(* IEC 61131-3 sources: repolevel_ST_code_completion/extract_code/轴控/FB105_轴控制集/FC11_设备状态, 3 files *)

(* ---- A03_气缸状态.st ---- *)
IF DI_取料上下气缸原点 AND DI_入料纠偏气缸原点 AND DI_翻板气缸原点 AND DI_左A包底气缸原点 AND DI_右B包底气缸原点 AND
	DI_上包底气缸原点 AND DI_出料推盒气缸原点 AND DI_包盒口升降气缸原点 AND DI_包盒口下压气缸原点 AND DI_推底板气缸原点 AND
	 DI_翻底板气缸原点 AND DI_模组吸底板气缸原点 THEN
	 b所有气缸原位OK:=TRUE;
	 ELSE
	 b所有气缸原位OK:=FALSE;
END_IF

IF NOT DO_取料气缸 AND NOT DO_纠偏气缸 AND NOT DO_挡料定位气缸 AND NOT DO_翻板气缸 AND NOT DO_侧压紧气缸 AND NOT DO_左A包底气缸 AND
	NOT DO_右B包底气缸 AND NOT DO_上包底气缸 AND NOT DO_下包底气缸 AND NOT DO_出料推盒气缸 AND NOT DO_包盒口升降气缸 AND
	NOT DO_包盒口下压气缸 AND NOT DO_翻底板气缸 AND NOT DO_推底板气缸 AND NOT DO_模组吸底板气缸 AND NOT DO_包边纠偏上下气缸 AND
	NOT DO_包边纠偏左右气缸 AND NOT DO_包边压料气缸 AND NOT DO_折边上托气缸 AND NOT DO_包边铲边气缸 AND NOT DO_吸底板真空 AND
	NOT DO_取面板真空 AND NOT DO_A模吸底板真空 AND NOT DO_A模吸面板真空 AND NOT DO_B模吸底板真空 AND NOT DO_B模吸面板真空 THEN
	b所有气缸关闭OK:=TRUE;
	ELSE
	b所有气缸关闭OK:=FALSE;
END_IF

(* ---- A04_初始化.st ---- *)
TON0(IN:= HMI_b初始化, PT:= T#3S, Q=> , ET=> );
TON1(IN:= HMI_b初始化, PT:= T#2S, Q=> , ET=> );
R_TRIG0(CLK:= TON0.Q AND b所有伺服使能OK AND b所有伺服总线通讯OK AND NOT b设备报警 AND b非急停手动模式 AND NOT b设备初始化中, Q=> );
R_TRIG1(CLK:= TON1.Q AND b所有伺服使能OK AND b所有伺服总线通讯OK AND NOT b设备报警 AND b非急停手动模式 AND NOT b设备初始化中, Q=> );

IF R_TRIG1.Q THEN
	b轴控初始化:=TRUE;
END_IF
TON4(IN:= b轴控初始化, PT:= T#0.3S, Q=> , ET=> );
IF TON4.Q THEN
	b轴控初始化:=FALSE;
END_IF

IF NOT DI_急停按钮 THEN
	i初始化步:=0;
	b设备初始化中:=FALSE;
	b调模A轴回零触发:=FALSE;
	b调模B轴回零触发:=FALSE;
	b送面料轴回零触发:=FALSE;
	b取面料轴回零触发:=FALSE;
	b横移A轴回零触发:=FALSE;
	b升降A轴回零触发:=FALSE;
	b横移B轴回零触发:=FALSE;
	b升降B轴回零触发:=FALSE;
	b出盒轴回零触发:=FALSE;
	b铲灰板轴回零触发:=FALSE;
	b包面纸轴回零触发:=FALSE;
	b上包底轴回零触发:=FALSE;
	b折边轴回零触发:=FALSE;
END_IF

CASE i初始化步 OF
	0:
	IF R_TRIG0.Q THEN
		b设备初始化中:=TRUE;
		i初始化步:=1;
	END_IF

	1:
	IF b设备初始化中 THEN
		b自动运行:=FALSE; b自动互锁:=FALSE;
		TON2(IN:= TRUE, PT:= T#0.2S, Q=> , ET=> );
		IF TON2.Q THEN
			TON2(IN:= FALSE,  );
			i初始化步:=5;
		END_IF

	END_IF

	5:

	IF b设备初始化中 THEN
		DO_取料气缸:=FALSE; DO_纠偏气缸:=FALSE; DO_挡料定位气缸:=FALSE; DO_翻板气缸:=FALSE; DO_侧压紧气缸:=FALSE;
		DO_左A包底气缸:=FALSE; DO_右B包底气缸:=FALSE; DO_上包底气缸:=FALSE; DO_下包底气缸:=FALSE; DO_出料推盒气缸:=FALSE;
		DO_包盒口升降气缸:=FALSE; DO_包盒口下压气缸:=FALSE; DO_翻底板气缸:=FALSE; DO_推底板气缸:=FALSE; DO_模组吸底板气缸:=FALSE;
		DO_包边纠偏上下气缸:=FALSE; DO_包边纠偏左右气缸:=FALSE; DO_包边压料气缸:=FALSE; DO_折边上托气缸:=FALSE;
        DO_包边铲边气缸:=FALSE; DO_吸底板真空:=FALSE; DO_取面板真空:=FALSE; DO_A模吸底板真空:=FALSE; DO_A模吸面板真空:=FALSE;
		DO_B模吸底板真空:=FALSE; DO_B模吸面板真空:=FALSE; DO_真空泵:=FALSE; DO_出料皮带电机:=FALSE;
		IF b所有气缸原位OK AND b所有气缸关闭OK THEN
			i初始化步:=10;
		END_IF
	END_IF

	10:
	IF b设备初始化中 THEN
		b调模A轴回零触发:=TRUE;
		b调模B轴回零触发:=TRUE;
		b送面料轴回零触发:=TRUE;
		b取面料轴回零触发:=TRUE;
		b横移A轴回零触发:=TRUE;
		b升降A轴回零触发:=TRUE;
		b横移B轴回零触发:=TRUE;
		b升降B轴回零触发:=TRUE;
		b出盒轴回零触发:=TRUE;
		b铲灰板轴回零触发:=TRUE;
		b包面纸轴回零触发:=TRUE;
		b上包底轴回零触发:=TRUE;
		b折边轴回零触发:=TRUE;
		TON3(IN:= TRUE, PT:= T#0.2S, Q=> , ET=> );
		IF TON3.Q AND b所有伺服静止中 THEN
			b调模A轴回零触发:=FALSE;
		    b调模B轴回零触发:=FALSE;
		    b送面料轴回零触发:=FALSE;
		    b取面料轴回零触发:=FALSE;
		    b横移A轴回零触发:=FALSE;
		    b升降A轴回零触发:=FALSE;
		    b横移B轴回零触发:=FALSE;
		    b升降B轴回零触发:=FALSE;
		    b出盒轴回零触发:=FALSE;
		    b铲灰板轴回零触发:=FALSE;
		    b包面纸轴回零触发:=FALSE;
		    b上包底轴回零触发:=FALSE;
		    b折边轴回零触发:=FALSE;
			TON3(IN:= FALSE,  );
			i初始化步:=15;
		END_IF

	END_IF

	15:
	IF b设备初始化中 THEN
		b设备初始化中:=FALSE;
		i初始化步:=0;
	END_IF
END_CASE

(* ---- FB11_设备状态.st ---- *)
PROGRAM FC11_设备状态
VAR
	fb_bFristScan: TON;

	TON0: TON;
	TON1: TON;
	TON2: TON;
	TON3: TON;
	TON4: TON;

	i初始化步: INT;

	R_TRIG0: R_TRIG;
	R_TRIG1: R_TRIG;

END_VAR

(*IO功能启用*)
//NET_IO_Cmd(SysWarnID:= , bError=> , nErrorID=> );

(*子程序调用*)
A01_输入映射();

A02_输出映射();

A03_气缸状态();

A04_初始化();

(*开机初始化*)
fb_bFristScan(IN:= b常闭, PT:= T#1S, Q=> , ET=> );
IF TIME_TO_REAL(fb_bFristScan.ET)>500 AND TIME_TO_REAL(fb_bFristScan.ET)<600 THEN
	b开机初始化:=TRUE;
	ELSE
	b开机初始化:=FALSE;
END_IF

IF NOT b常通 THEN
	b开机第一次启动:=TRUE;
	ELSE
	b开机第一次启动:=FALSE;
END_IF
IF b开机第一次启动 OR b常通 THEN
	b常通:=TRUE;
	ELSE
	b常通:=FALSE;
END_IF
(*
IF EtherCAT_Master_Leadshine.xConfigFinished AND EtherCAT_Master_Leadshine.xDistributedClockInSync AND
   NOT EtherCAT_Master_Leadshine.xError AND NOT b常闭 THEN
	b开机初始化:=TRUE;
	ELSE
	b开机初始化:=FALSE;
END_IF
*)

(*状态判定*)
IF DI_急停按钮 AND NOT HMI_b手动模式0自动模式1 THEN
	b非急停手动模式:=TRUE;
	ELSE
	b非急停手动模式:=FALSE;
END_IF
IF DI_急停按钮 AND HMI_b手动模式0自动模式1 THEN
	b非急停自动模式:=TRUE;
	ELSE
	b非急停自动模式:=FALSE;
END_IF
